// TIA Portal V17 export
TYPE "Recipe"
   STRUCT
      "Name" : String[20] := 'Standard';
      Speed : Real := 1.5;
      Limits : Struct
         Min : Int;
         Max : Int := 100;
      END_STRUCT;
   END_STRUCT;
END_TYPE
